// TwinCAT 3 PLC project Puller_PLC
// ProgramVersion: 3.1.4024.0
// libraries:
//   Tc2_Standard, * (Beckhoff Automation GmbH)
//   Tc2_System, * (Beckhoff Automation GmbH)
//   Tc3_Module, * (Beckhoff Automation GmbH)
// project tree:
//   DUTs/01_炉体单元/ ST_DomeCharmber.TcDUT (not stored), ST_MainCharmber.TcDUT (not stored), ST_PullCharmber.TcDUT
//   DUTs/02_真空压力单元/ ST_ArGas.TcDUT, ST_BackBlowSys.TcDUT, ST_PressureMeasure.TcDUT, ST_PumpSys.TcDUT
//   DUTs/ ST_CrucibleLiftSys.TcDUT, ST_HmiIVar.TcDUT, ST_IngotPrevent.TcDUT, ST_MagnetControl.TcDUT, ST_MagnetLiftSys.TcDUT, ST_PowerHeaterSys.TcDUT, ST_SeedLiftSys.TcDUT, ST_SystemVar.TcDUT, ST_TempMeasure.TcDUT, ST_GateValve.TcDUT
//   GVLs/ GVL_Pulller.TcGVL
//   / PlcTask.TcTTO
//   POUs/FB_APS_Prog/ FB_APS_Prog.TcPOU, ST_APS_Data.TcDUT
//   POUs/ MAIN.TcPOU
// real-time tasks:
//   TASK PlcTask: cycle T#10ms, priority 20, ADS port 350

CONFIGURATION Puller_PLC
    RESOURCE PLC ON TwinCAT3
        TASK PlcTask(INTERVAL := T#10ms, PRIORITY := 20);
        PROGRAM MAIN WITH PlcTask : MAIN;
    END_RESOURCE
END_CONFIGURATION

// ---- DUTs/01_炉体单元/ST_PullCharmber.TcDUT
TYPE ST_PullCharmber :
STRUCT
END_STRUCT
END_TYPE

// ---- DUTs/02_真空压力单元/ST_ArGas.TcDUT
TYPE ST_ArGas :
STRUCT
	boAr1_OPen:BOOL;
	boAr2_OPen:BOOL;
	boAr3_Open:BOOL;
	nAr1FlowValva:INT;
	nAr2FlowValva:INT;
	nAr3FlowValva:INT;

END_STRUCT
END_TYPE

// ---- DUTs/02_真空压力单元/ST_BackBlowSys.TcDUT
TYPE ST_BackBlowSys :
STRUCT
END_STRUCT
END_TYPE

// ---- DUTs/02_真空压力单元/ST_PressureMeasure.TcDUT
TYPE ST_PressureMeasure:
STRUCT
	fiPullChumberVac:REAL;
	fiMainChumberVac:REAL;
	fiGrownPressVac:REAL;
END_STRUCT
END_TYPE

// ---- DUTs/02_真空压力单元/ST_PumpSys.TcDUT
TYPE ST_PumpSys :
STRUCT
	boAuxPump_On:BOOL;
	boAuxPump_Off:BOOL;
	boAuxPumpValve_On:BOOL;
	boMainPump_On:BOOL;
	boMainPump_Off:BOOL;
	boMainPumpValve_On:BOOL;
	boMainPumpValve_Off:BOOL;
	biMainPumpErr:BOOL;
END_STRUCT
END_TYPE

// ---- DUTs/ST_CrucibleLiftSys.TcDUT
TYPE ST_CrucibleLiftSys :
STRUCT
END_STRUCT
END_TYPE

// ---- DUTs/ST_HmiIVar.TcDUT
TYPE ST_HmiIVar :
STRUCT
	bApsOnBtn:BOOL;
	bApsOnLamp:BOOL;//12
	
END_STRUCT
END_TYPE

// ---- DUTs/ST_IngotPrevent.TcDUT
TYPE ST_IngotPrevent :
STRUCT
	biSnIngotPrevent_Forward:BOOL;
	biSnIngotPrevent_Back:BOOL;
	BoCylIngotPrevent_Forward:BOOL;
	BoCylIngotPrevent_Back:BOOL;
	biSnIngotPreventBtn_Forward:BOOL;
	biSnIngotPreventBtn_Back:BOOL;
END_STRUCT
END_TYPE

// ---- DUTs/ST_MagnetControl.TcDUT
TYPE ST_MagnetControl :
STRUCT
END_STRUCT
END_TYPE

// ---- DUTs/ST_MagnetLiftSys.TcDUT
TYPE ST_MagnetLiftSys :
STRUCT
END_STRUCT
END_TYPE

// ---- DUTs/ST_PowerHeaterSys.TcDUT
TYPE ST_PowerHeaterSys :
STRUCT
END_STRUCT
END_TYPE

// ---- DUTs/ST_SeedLiftSys.TcDUT
TYPE ST_SeedLiftSys :
STRUCT
END_STRUCT
END_TYPE

// ---- DUTs/ST_SystemVar.TcDUT
TYPE ST_SystemVar :
STRUCT
	bNoProcessStu:BOOL;
END_STRUCT
END_TYPE

// ---- DUTs/ST_TempMeasure.TcDUT
TYPE ST_TempMeasure :
STRUCT
END_STRUCT
END_TYPE

// ---- DUTs/ST_GateValve.TcDUT
TYPE ST_GateValve :
STRUCT
	biSnGateValve_Close:BOOL;
	biSnGateValve_Open:BOOL;
	boCylGateValve_Close:BOOL;
	boCylGateValve_Open:BOOL;
END_STRUCT
END_TYPE

// ---- POUs/FB_APS_Prog/ST_APS_Data.TcDUT
TYPE ST_APS_Data :
STRUCT	
	bArPurgeProcessStart:BOOL;
	bArPurgeProcessing:BOOL;
	nAr1PurgeFlow:INT;
	nArPurgeSetCount:INT:=3;
	nArPurgeCurrentCount:INT;
	nUpperPressureSet:INT:=1000;
	nLowerPressureSet:INT:=50;
	nCurrentPressure:INT;
	nPull_MainGapPressureSet:INT;
	nStepNo:INT;
	tStepDelayTime:ton;
END_STRUCT
END_TYPE

// ---- GVLs/GVL_Pulller.TcGVL
//{attribute 'qualified_only'}
VAR_GLOBAL
	stArGas:ST_ArGas;
	stIngotPrevent:ST_IngotPrevent;
	stPressureMeasure:ST_PressureMeasure;
	stPumpSys:ST_PumpSys;
	stGateValve:St_GateValve;
	stHmiVar:ST_HmiIVar;
	stSystemVar:St_SystemVar;
END_VAR

// ---- POUs/MAIN.TcPOU
PROGRAM MAIN
VAR
	fbAPS_Prog:FB_APS_Prog;
END_VAR

fbAPS_Prog();

END_PROGRAM

// ---- POUs/FB_APS_Prog/FB_APS_Prog.TcPOU
FUNCTION_BLOCK FB_APS_Prog
VAR_INPUT
	ApsFunctionEnable:BOOL;
END_VAR
VAR_OUTPUT
END_VAR
VAR
	_stAPSData:ST_APS_Data;	
END_VAR

IF ApsFunctionEnable THEN
{region"APS启动"}
//APS工艺流程启动
	IF stGateValve.biSnGateValve_Close
	AND stHmiVar.bApsOnBtn 
	AND stSystemVar.bNoProcessStu 
	AND NOT _stAPSData.bArPurgeProcessing THEN
		_stAPSData.bArPurgeProcessStart:=TRUE;		
	END_IF
		 
//APS工艺流程中...
	IF _stAPSData.bArPurgeProcessStart THEN
		_stAPSData.bArPurgeProcessing:=TRUE;
		_stAPSData.bArPurgeProcessStart:=FALSE;
		_stAPSData.nStepNo:=10;
	END_IF
{endregion}
	 
{region"APS自动流程"}
//APS自动清扫流程启动
	CASE _stAPSData.nStepNo OF
		10://APS启动初始化（AUX真空泵开启,Ar1流量设定）
			 stPumpSys.boAuxPumpValve_On:=FALSE;
			 stPumpSys.boAuxPump_On:=TRUE;
			 stArGas.nAr1FlowValva:=_stAPSData.nAr1PurgeFlow;
			_stAPSData.tStepDelayTime(IN:=TRUE , PT:=T#5S );
			IF _stAPSData.tStepDelayTime.Q THEN 
				_stAPSData.nStepNo:=30;
				_stAPSData.tStepDelayTime(IN:=FALSE );
			END_IF
		(*20://AUX真空泵开启
			stPumpSys.boAuxPump_On:=TRUE;
			_stAPSData.tStepDelayTime(IN:=TRUE , PT:=T#5S );
			IF _stAPSData.tStepDelayTime.Q THEN 
				_stAPSData.nStepNo:=30;
				_stAPSData.tStepDelayTime(IN:=FALSE );
			END_IF*)
		30://AUX真空阀门开启
			stPumpSys.boAuxPumpValve_On:=TRUE;
			_stAPSData.tStepDelayTime(IN:=TRUE , PT:=T#2S );
			IF _stAPSData.tStepDelayTime.Q  THEN 
				_stAPSData.nStepNo:=40;
				_stAPSData.tStepDelayTime(IN:=FALSE );
			END_IF	
		40://真空压力达到下限值
			IF stPressureMeasure.fiPullChumberVac < _stAPSData.nLowerPressureSet THEN 
				_stAPSData.nStepNo:=50;
			END_IF	
		50://AUX真空阀关闭
			stPumpSys.boAuxPumpValve_On:=FALSE;
			_stAPSData.tStepDelayTime(IN:=TRUE , PT:=T#1S );
			IF _stAPSData.tStepDelayTime.Q  THEN
				IF _stAPSData.nArPurgeSetCount=0 THEN
				_stAPSData.nStepNo:=120;
				ELSE
				_stAPSData.nStepNo:=60;	 
				END_IF 
				_stAPSData.tStepDelayTime(IN:=FALSE );
			END_IF
		60://Ar1阀门开启
			stArGas.boAr1_OPen:=TRUE;
			_stAPSData.tStepDelayTime(IN:=TRUE , PT:=T#1S );
			IF _stAPSData.tStepDelayTime.Q  THEN 
				_stAPSData.nStepNo:=70;
				_stAPSData.tStepDelayTime(IN:=FALSE );
			END_IF
		70://真空压力值达到上限
			IF stPressureMeasure.fiPullChumberVac> _stAPSData.nUpperPressureSet THEN 
				_stAPSData.nStepNo:=80;
			END_IF		 
		80://Ar1阀门关闭
			stArGas.boAr1_OPen:=FALSE;
			_stAPSData.tStepDelayTime(IN:=TRUE , PT:=T#1S );
			IF _stAPSData.tStepDelayTime.Q  THEN 
				_stAPSData.nStepNo:=90;
				_stAPSData.tStepDelayTime(IN:=FALSE );
			END_IF	
		90://AUX真空阀门开启
			stPumpSys.boAuxPumpValve_On:=TRUE;
			_stAPSData.tStepDelayTime(IN:=TRUE , PT:=T#2S );
			IF _stAPSData.tStepDelayTime.Q  THEN 
				_stAPSData.nStepNo:=100;
				_stAPSData.tStepDelayTime(IN:=FALSE );
			END_IF	
		
		100://真空压力达到下限值
			IF stPressureMeasure.fiPullChumberVac <= _stAPSData.nLowerPressureSet THEN 	
				_stAPSData.nStepNo:=110;
			END_IF				 
		110://AUX真空阀关闭
			stPumpSys.boAuxPumpValve_On:=FALSE;
			_stAPSData.tStepDelayTime(IN:=TRUE , PT:=T#1S );
			IF _stAPSData.tStepDelayTime.Q  THEN
				_stAPSData.nArPurgeCurrentCount:=_stAPSData.nArPurgeCurrentCount+1;
				IF _stAPSData.nArPurgeCurrentCount>= _stAPSData.nArPurgeSetCount THEN
					_stAPSData.nStepNo:=120;
				ELSE
					_stAPSData.nStepNo:=60;	 
				END_IF					 
			END_IF
		120://APS自动流程结束
			_stAPSData.bArPurgeProcessStart:=FALSE;
			_stAPSData.bArPurgeProcessing:=FALSE;
			_stAPSData.nArPurgeCurrentCount:=0;
			_stAPSData.nStepNo:=0;	
			stPumpSys.boAuxPump_On:=FALSE;
	END_CASE

{endregion}	
END_IF

//APS系统流程关闭
IF stGateValve.biSnGateValve_Open
	OR NOT stSystemVar.bNoProcessStu 
	OR NOT ApsFunctionEnable THEN
		_stAPSData.bArPurgeProcessStart:=FALSE;
		_stAPSData.bArPurgeProcessing:=FALSE;
		_stAPSData.nArPurgeCurrentCount:=0;
		_stAPSData.nStepNo:=0;
END_IF

END_FUNCTION_BLOCK
